// TIA Portal V19 export
TYPE "TetraPakV50_IO"
TITLE = TPV50_9_IO
// DEVICEID : 9
//  VENDOR : IFM on behalf of Tetra Pak
//  DATE: 27.12.2023 
// 
//  Comment : TP V50 IO Interface
   STRUCT
      IN : Struct
         Address : Int;   // First Byte address of 4 byte address space
         Pulse : Bool;   // Trigger one clean pulse on SV 1
         SV_1 : Bool;   // Trigger solenoid valve 1 for main valve activation
         Wink : Bool;   // Visual indication for locating the unit
      END_STRUCT;
      OUT : Struct
         ValvePosition : Real;   // Current Valve position (0 to 720 * 0.1)
         ErrorStatus : Byte;   // See Block Comment
         ValveState : Bool;   // Current Valve state
         Main : Bool;   // Main energised Position
         DE_EN : Bool;   // De-energised
         O_DI4 : Bool;   // Output signal status Pin 4
         O_DI2 : Bool;   // Output signal status Pin 2
         O_DA : Bool;   // Output device recognised
         O_DE : Bool;   // Output device error event has appeared
         O_PQ : Bool;   // Output port qualifer proces data valid
      END_STRUCT;
      IN_OUT : Struct
         HMI_INFO : Int;
         HMI_CMD : Int;
      END_STRUCT;
   END_STRUCT;
END_TYPE
